(* IEC 61131-3 sources: plc_generation_empirical_study/datasets/task_bank_c06_reverse_bounded_runtime_v0_3/tasks/C06_V17_lean_composite/negative_control, 1 file *)

(* ---- NC1.st ---- *)
FUNCTION_BLOCK C06_V17_lean_composite
VAR_INPUT
    A_AutoMode : BOOL;
    A_AutoDemand : BOOL;
    A_ManualDemand : BOOL;
    A_SafetyOK : BOOL;
    A_Inhibit : BOOL;
    B_Inspected : BOOL;
    B_Rejected : BOOL;
    B_Reset : BOOL;
    B_WindowSize : INT;
    B_RejectLimit : INT;
    SubsystemBEnable : BOOL;
    CrossReset : BOOL;
END_VAR
VAR_OUTPUT
    A_Command : BOOL;
    A_Blocked : BOOL;
    B_WindowCount : INT;
    B_RejectCount : INT;
    B_LockedOut : BOOL;
    B_WindowComplete : BOOL;
    CrossReady : BOOL;
    CrossBlocked : BOOL;
END_VAR
VAR
    B_PrevInspected : BOOL := FALSE;
END_VAR

A_Command := ((A_AutoMode AND A_AutoDemand) OR ((NOT A_AutoMode) AND A_ManualDemand))
           AND A_SafetyOK AND (NOT A_Inhibit);
A_Blocked := ((A_AutoMode AND A_AutoDemand) OR ((NOT A_AutoMode) AND A_ManualDemand))
           AND ((NOT A_SafetyOK) OR A_Inhibit);

IF CrossReset THEN
    CrossReady := FALSE;
ELSIF A_Command THEN
    CrossReady := TRUE;
END_IF;
CrossBlocked := FALSE;

IF SubsystemBEnable AND CrossReady THEN
    B_WindowComplete := FALSE;
    IF B_Reset THEN
        B_WindowCount := 0;
        B_RejectCount := 0;
        B_LockedOut := FALSE;
    ELSIF (NOT B_LockedOut) AND B_Inspected AND (NOT B_PrevInspected) THEN
        B_WindowCount := B_WindowCount + 1;
        IF B_Rejected THEN
            B_RejectCount := B_RejectCount + 1;
        END_IF;
        IF B_WindowCount >= B_WindowSize THEN
            IF B_RejectCount > B_RejectLimit THEN
                B_LockedOut := TRUE;
            END_IF;
            B_WindowCount := 0;
            B_RejectCount := 0;
            B_WindowComplete := TRUE;
        END_IF;
    END_IF;
    B_PrevInspected := B_Inspected;
ELSE
    B_WindowCount := 0;
    B_RejectCount := 0;
    B_LockedOut := FALSE;
    B_WindowComplete := FALSE;
END_IF;

END_FUNCTION_BLOCK
